// TIA Portal V20 export
TYPE "typeIntConditionHmiInterface"
// stored: Access Published, Namespace Unit1.Em1
   STRUCT
      Actuator_08 { S7_SetPoint := 'True'} : "LER_typeAxisActuatorCondition";   // AnodeNgBoxLockUpDown
      Actuator_09 { S7_SetPoint := 'True'} : "LER_typeAxisActuatorCondition";   // AnodeMaintenanceMovingFixFrontFwdBwd
      Actuator_10 { S7_SetPoint := 'True'} : "LER_typeAxisActuatorCondition";   // AnodeMaintenanceMovingFixFrontFwdBwd
      Actuator_11 { S7_SetPoint := 'True'} : "LER_typeAxisActuatorCondition";   // AnodeNgBoxLockUpDown
      Actuator_12 { S7_SetPoint := 'True'} : "LER_typeAxisActuatorCondition";   // AnodeMaintenanceMovingFixFrontFwdBwd
      Actuator_13 { S7_SetPoint := 'True'} : "LER_typeAxisActuatorCondition";   // AnodeNgBoxLockUpDown
      Actuator_14 { S7_SetPoint := 'True'} : "LER_typeAxisActuatorCondition";   // AnodeMaintenanceMovingFixFrontFwdBwd
   END_STRUCT;
END_TYPE
